// TIA Portal V19 export
VAR_GLOBAL   // PLC tag table "Encoder"
END_VAR
